// Mitsubishi GX Works2 project: NIAP1854_1000_RC-1M_5B_R3   PLC: FX3S

PROGRAM MAIN
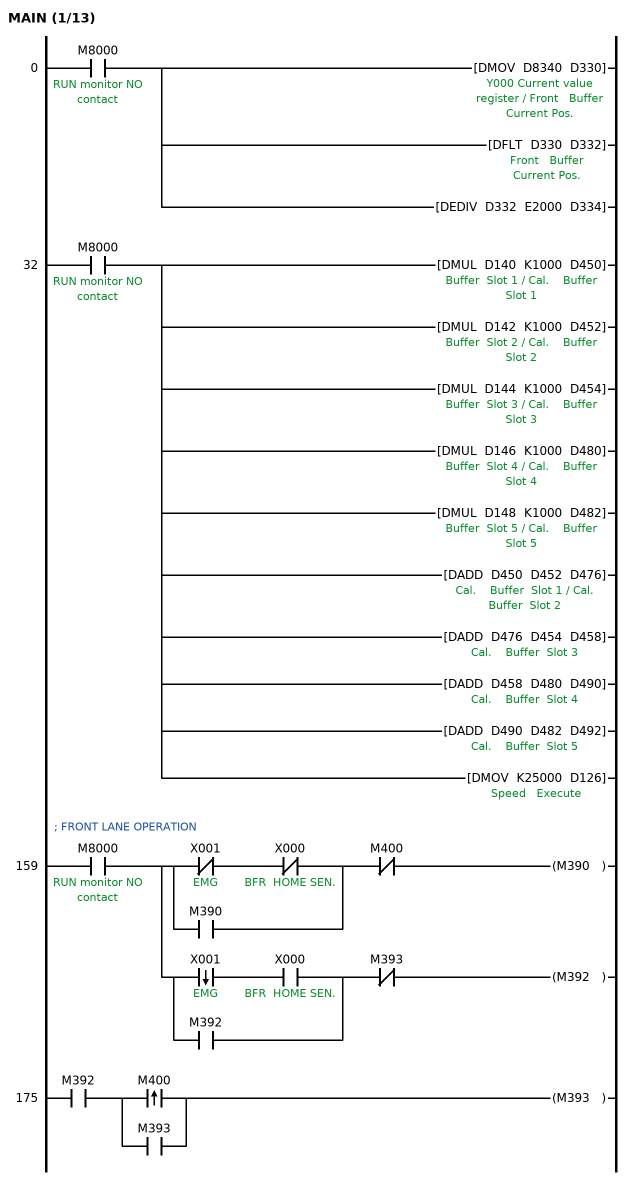
0     LD      M8000  ; RUN monitor NO contact
      DMOV    D8340 D330  ; Y000 Current value register / Front   Buffer  Current Pos.
      DFLT    D330 D332
      DEDIV   D332 E2000 D334
32    LD      M8000  ; RUN monitor NO contact
      DMUL    D140 K1000 D450  ; Buffer  Slot 1 / Cal.    Buffer  Slot 1
      DMUL    D142 K1000 D452  ; Buffer  Slot 2 / Cal.    Buffer  Slot 2
      DMUL    D144 K1000 D454  ; Buffer  Slot 3 / Cal.    Buffer  Slot 3
      DMUL    D146 K1000 D480  ; Buffer  Slot 4 / Cal.    Buffer  Slot 4
      DMUL    D148 K1000 D482  ; Buffer  Slot 5 / Cal.    Buffer  Slot 5
      DADD    D450 D452 D476
      DADD    D476 D454 D458
      DADD    D458 D480 D490
      DADD    D490 D482 D492
      DMOV    K25000 D126  ; Speed   Execute
; FRONT LANE OPERATION
159   LD      M8000  ; RUN monitor NO contact
      MPS
      LDI     X001  ; EMG
      ANI     X000  ; BFR  HOME SEN.
      OR      M390
      ANB
      ANI     M400
      OUT     M390
      MPP
      LDF     X001  ; EMG
      AND     X000  ; BFR  HOME SEN.
      OR      M392
      ANB
      ANI     M393
      OUT     M392
175   LD      M392
      LDP     M400
      OR      M393
      ANB
      OUT     M393
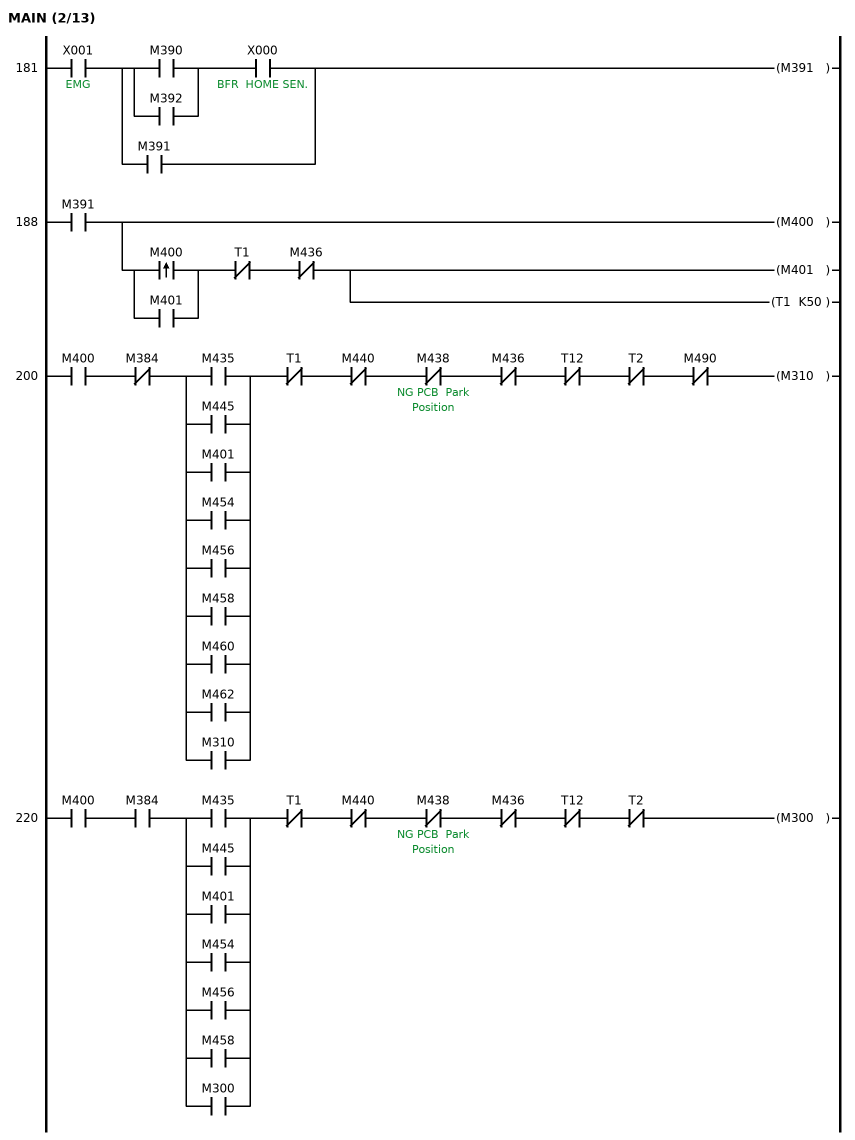
181   LD      X001  ; EMG
      LD      M390
      OR      M392
      AND     X000  ; BFR  HOME SEN.
      OR      M391
      ANB
      OUT     M391
188   LD      M391
      OUT     M400
      LDP     M400
      OR      M401
      ANB
      ANI     T1
      ANI     M436
      OUT     M401
      OUT     T1 K50
200   LD      M400
      ANI     M384
      LD      M435
      OR      M445
      OR      M401
      OR      M454
      OR      M456
      OR      M458
      OR      M460
      OR      M462
      OR      M310
      ANB
      ANI     T1
      ANI     M440
      ANI     M438  ; NG PCB  Park    Position
      ANI     M436
      ANI     T12
      ANI     T2
      ANI     M490
      OUT     M310
220   LD      M400
      AND     M384
      LD      M435
      OR      M445
      OR      M401
      OR      M454
      OR      M456
      OR      M458
      OR      M300
      ANB
      ANI     T1
      ANI     M440
      ANI     M438  ; NG PCB  Park    Position
      ANI     M436
      ANI     T12
      ANI     T2
      OUT     M300
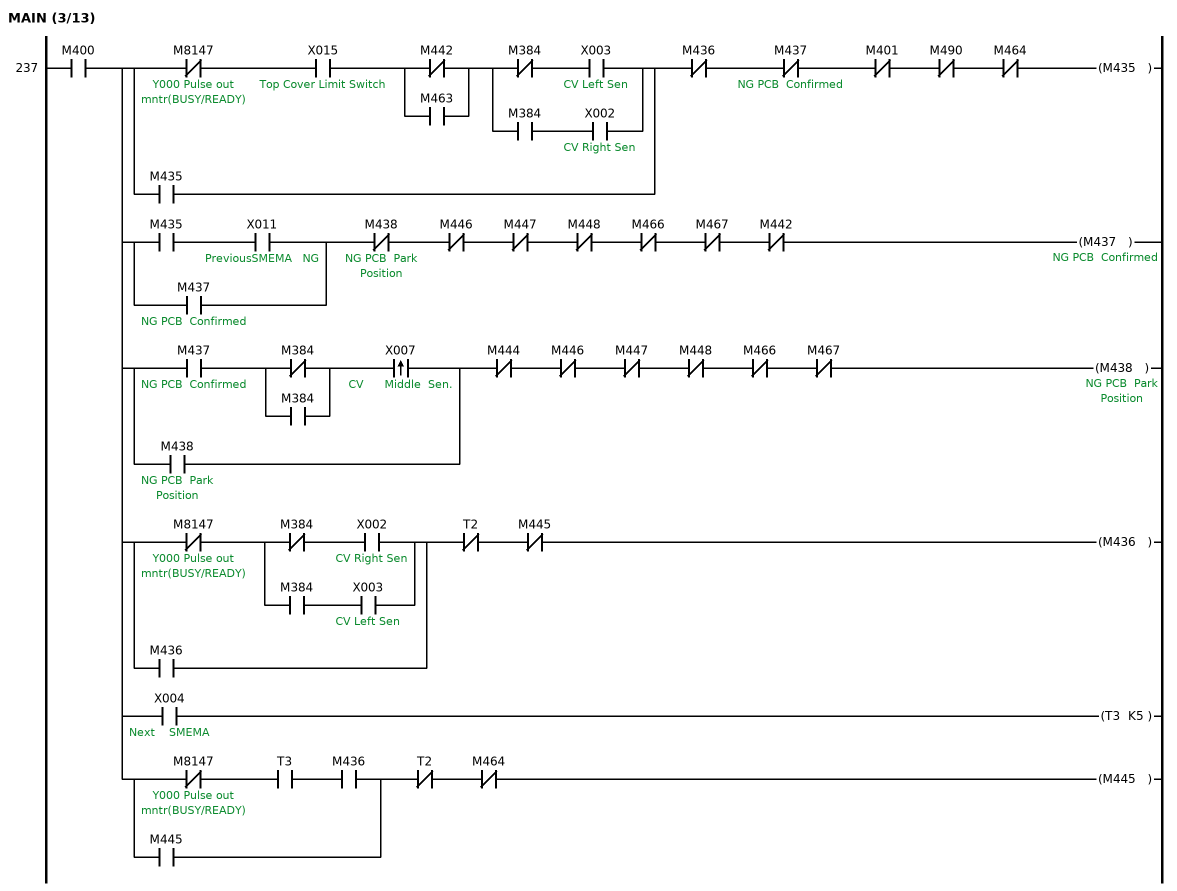
237   LD      M400
      MPS
      LDI     M8147  ; Y000 Pulse out mntr(BUSY/READY)
      AND     X015  ; Top Cover Limit Switch
      LDI     M442
      OR      M463
      ANB
      LDI     M384
      AND     X003  ; CV Left Sen
      LD      M384
      AND     X002  ; CV Right Sen
      ORB
      ANB
      OR      M435
      ANB
      ANI     M436
      ANI     M437  ; NG PCB  Confirmed
      ANI     M401
      ANI     M490
      ANI     M464
      OUT     M435
      MRD
      LD      M435
      AND     X011  ; PreviousSMEMA   NG
      OR      M437  ; NG PCB  Confirmed
      ANB
      ANI     M438  ; NG PCB  Park    Position
      ANI     M446
      ANI     M447
      ANI     M448
      ANI     M466
      ANI     M467
      ANI     M442
      OUT     M437  ; NG PCB  Confirmed
      MRD
      LD      M437  ; NG PCB  Confirmed
      LDI     M384
      OR      M384
      ANB
      ANDP    X007  ; CV      Middle  Sen.
      OR      M438  ; NG PCB  Park    Position
      ANB
      ANI     M444
      ANI     M446
      ANI     M447
      ANI     M448
      ANI     M466
      ANI     M467
      OUT     M438  ; NG PCB  Park    Position
      MRD
      LDI     M8147  ; Y000 Pulse out mntr(BUSY/READY)
      LDI     M384
      AND     X002  ; CV Right Sen
      LD      M384
      AND     X003  ; CV Left Sen
      ORB
      ANB
      OR      M436
      ANB
      ANI     T2
      ANI     M445
      OUT     M436
      MRD
      AND     X004  ; Next    SMEMA
      OUT     T3 K5
      MPP
      LDI     M8147  ; Y000 Pulse out mntr(BUSY/READY)
      AND     T3
      AND     M436
      OR      M445
      ANB
      ANI     T2
      ANI     M464
      OUT     M445
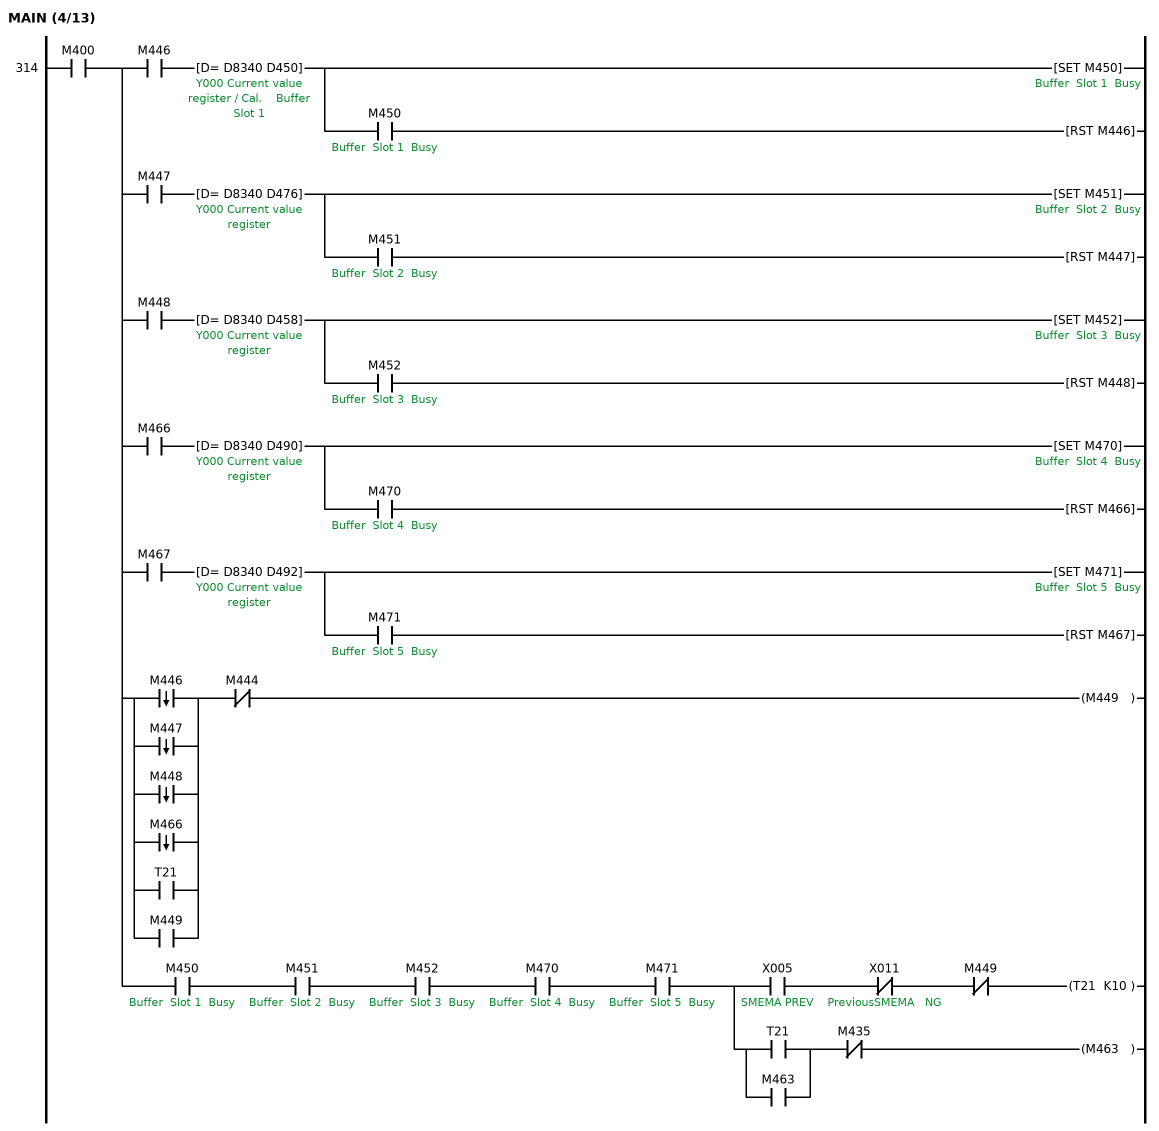
314   LD      M400
      MPS
      AND     M446
      ANDD=   D8340 D450  ; Y000 Current value register / Cal.    Buffer  Slot 1
      SET     M450  ; Buffer  Slot 1  Busy
      AND     M450  ; Buffer  Slot 1  Busy
      RST     M446
      MRD
      AND     M447
      ANDD=   D8340 D476  ; Y000 Current value register
      SET     M451  ; Buffer  Slot 2  Busy
      AND     M451  ; Buffer  Slot 2  Busy
      RST     M447
      MRD
      AND     M448
      ANDD=   D8340 D458  ; Y000 Current value register
      SET     M452  ; Buffer  Slot 3  Busy
      AND     M452  ; Buffer  Slot 3  Busy
      RST     M448
      MRD
      AND     M466
      ANDD=   D8340 D490  ; Y000 Current value register
      SET     M470  ; Buffer  Slot 4  Busy
      AND     M470  ; Buffer  Slot 4  Busy
      RST     M466
      MRD
      AND     M467
      ANDD=   D8340 D492  ; Y000 Current value register
      SET     M471  ; Buffer  Slot 5  Busy
      AND     M471  ; Buffer  Slot 5  Busy
      RST     M467
      MRD
      LDF     M446
      ORF     M447
      ORF     M448
      ORF     M466
      OR      T21
      OR      M449
      ANB
      ANI     M444
      OUT     M449
      MPP
      AND     M450  ; Buffer  Slot 1  Busy
      AND     M451  ; Buffer  Slot 2  Busy
      AND     M452  ; Buffer  Slot 3  Busy
      AND     M470  ; Buffer  Slot 4  Busy
      AND     M471  ; Buffer  Slot 5  Busy
      MPS
      AND     X005  ; SMEMA PREV
      ANI     X011  ; PreviousSMEMA   NG
      ANI     M449
      OUT     T21 K10
      MPP
      LD      T21
      OR      M463
      ANB
      ANI     M435
      OUT     M463
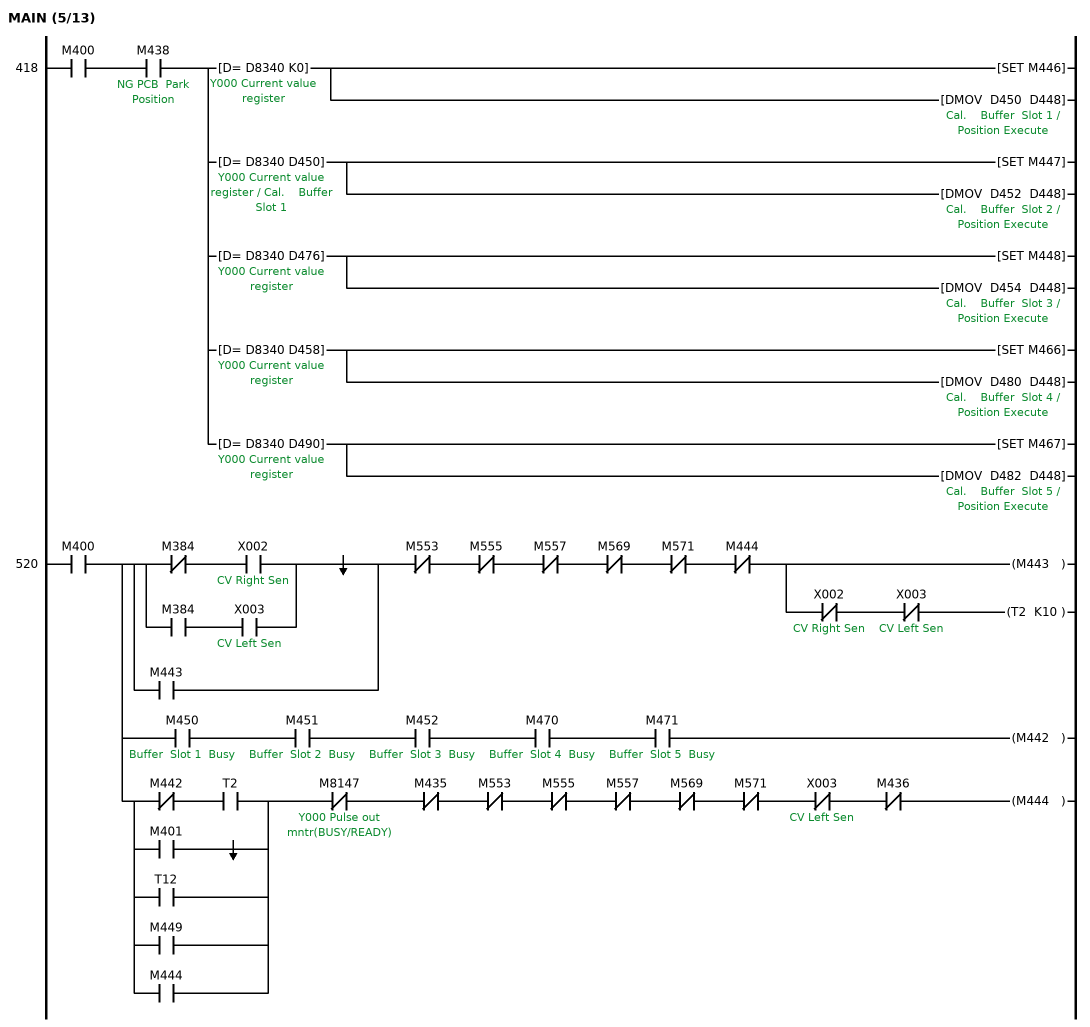
418   LD      M400
      AND     M438  ; NG PCB  Park    Position
      MPS
      ANDD=   D8340 K0  ; Y000 Current value register
      SET     M446
      DMOV    D450 D448  ; Position Execute
      MRD
      ANDD=   D8340 D450  ; Y000 Current value register / Cal.    Buffer  Slot 1
      SET     M447
      DMOV    D452 D448
      MRD
      ANDD=   D8340 D476  ; Y000 Current value register
      SET     M448
      DMOV    D454 D448
      MRD
      ANDD=   D8340 D458  ; Y000 Current value register
      SET     M466
      DMOV    D480 D448
      MPP
      ANDD=   D8340 D490  ; Y000 Current value register
      SET     M467
      DMOV    D482 D448
520   LD      M400
      MPS
      LDI     M384
      AND     X002  ; CV Right Sen
      LD      M384
      AND     X003  ; CV Left Sen
      ORB
      MEF
      OR      M443
      ANB
      ANI     M553
      ANI     M555
      ANI     M557
      ANI     M569
      ANI     M571
      ANI     M444
      OUT     M443
      ANI     X002  ; CV Right Sen
      ANI     X003  ; CV Left Sen
      OUT     T2 K10
      MRD
      AND     M450  ; Buffer  Slot 1  Busy
      AND     M451  ; Buffer  Slot 2  Busy
      AND     M452  ; Buffer  Slot 3  Busy
      AND     M470  ; Buffer  Slot 4  Busy
      AND     M471  ; Buffer  Slot 5  Busy
      OUT     M442
      MPP
      LDI     M442
      AND     T2
      LD      M401
      MEF
      ORB
      OR      T12
      OR      M449
      OR      M444
      ANB
      ANI     M8147  ; Y000 Pulse out mntr(BUSY/READY)
      ANI     M435
      ANI     M553
      ANI     M555
      ANI     M557
      ANI     M569
      ANI     M571
      ANI     X003  ; CV Left Sen
      ANI     M436
      OUT     M444
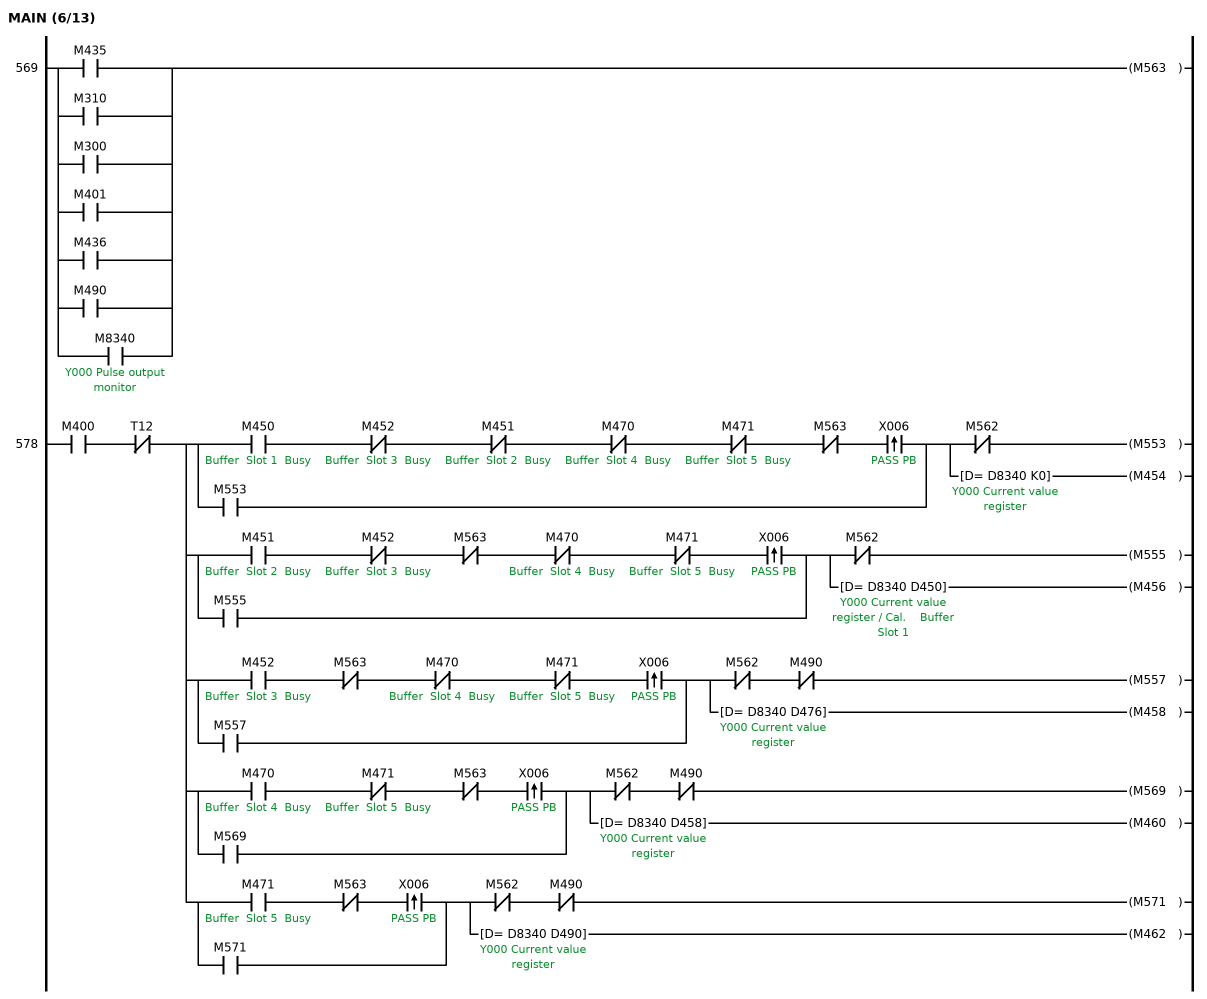
569   LD      M435
      OR      M310
      OR      M300
      OR      M401
      OR      M436
      OR      M490
      OR      M8340  ; Y000 Pulse output monitor
      OUT     M563
578   LD      M400
      ANI     T12
      MPS
      LD      M450  ; Buffer  Slot 1  Busy
      ANI     M452  ; Buffer  Slot 3  Busy
      ANI     M451  ; Buffer  Slot 2  Busy
      ANI     M470  ; Buffer  Slot 4  Busy
      ANI     M471  ; Buffer  Slot 5  Busy
      ANI     M563
      ANDP    X006  ; PASS PB
      OR      M553
      ANB
      MPS
      ANI     M562
      OUT     M553
      MPP
      ANDD=   D8340 K0  ; Y000 Current value register
      OUT     M454
      MRD
      LD      M451  ; Buffer  Slot 2  Busy
      ANI     M452  ; Buffer  Slot 3  Busy
      ANI     M563
      ANI     M470  ; Buffer  Slot 4  Busy
      ANI     M471  ; Buffer  Slot 5  Busy
      ANDP    X006  ; PASS PB
      OR      M555
      ANB
      MPS
      ANI     M562
      OUT     M555
      MPP
      ANDD=   D8340 D450  ; Y000 Current value register / Cal.    Buffer  Slot 1
      OUT     M456
      MRD
      LD      M452  ; Buffer  Slot 3  Busy
      ANI     M563
      ANI     M470  ; Buffer  Slot 4  Busy
      ANI     M471  ; Buffer  Slot 5  Busy
      ANDP    X006  ; PASS PB
      OR      M557
      ANB
      MPS
      ANI     M562
      ANI     M490
      OUT     M557
      MPP
      ANDD=   D8340 D476  ; Y000 Current value register
      OUT     M458
      MRD
      LD      M470  ; Buffer  Slot 4  Busy
      ANI     M471  ; Buffer  Slot 5  Busy
      ANI     M563
      ANDP    X006  ; PASS PB
      OR      M569
      ANB
      MPS
      ANI     M562
      ANI     M490
      OUT     M569
      MPP
      ANDD=   D8340 D458  ; Y000 Current value register
      OUT     M460
      MPP
      LD      M471  ; Buffer  Slot 5  Busy
      ANI     M563
      ANDP    X006  ; PASS PB
      OR      M571
      ANB
      MPS
      ANI     M562
      ANI     M490
      OUT     M571
      MPP
      ANDD=   D8340 D490  ; Y000 Current value register
      OUT     M462
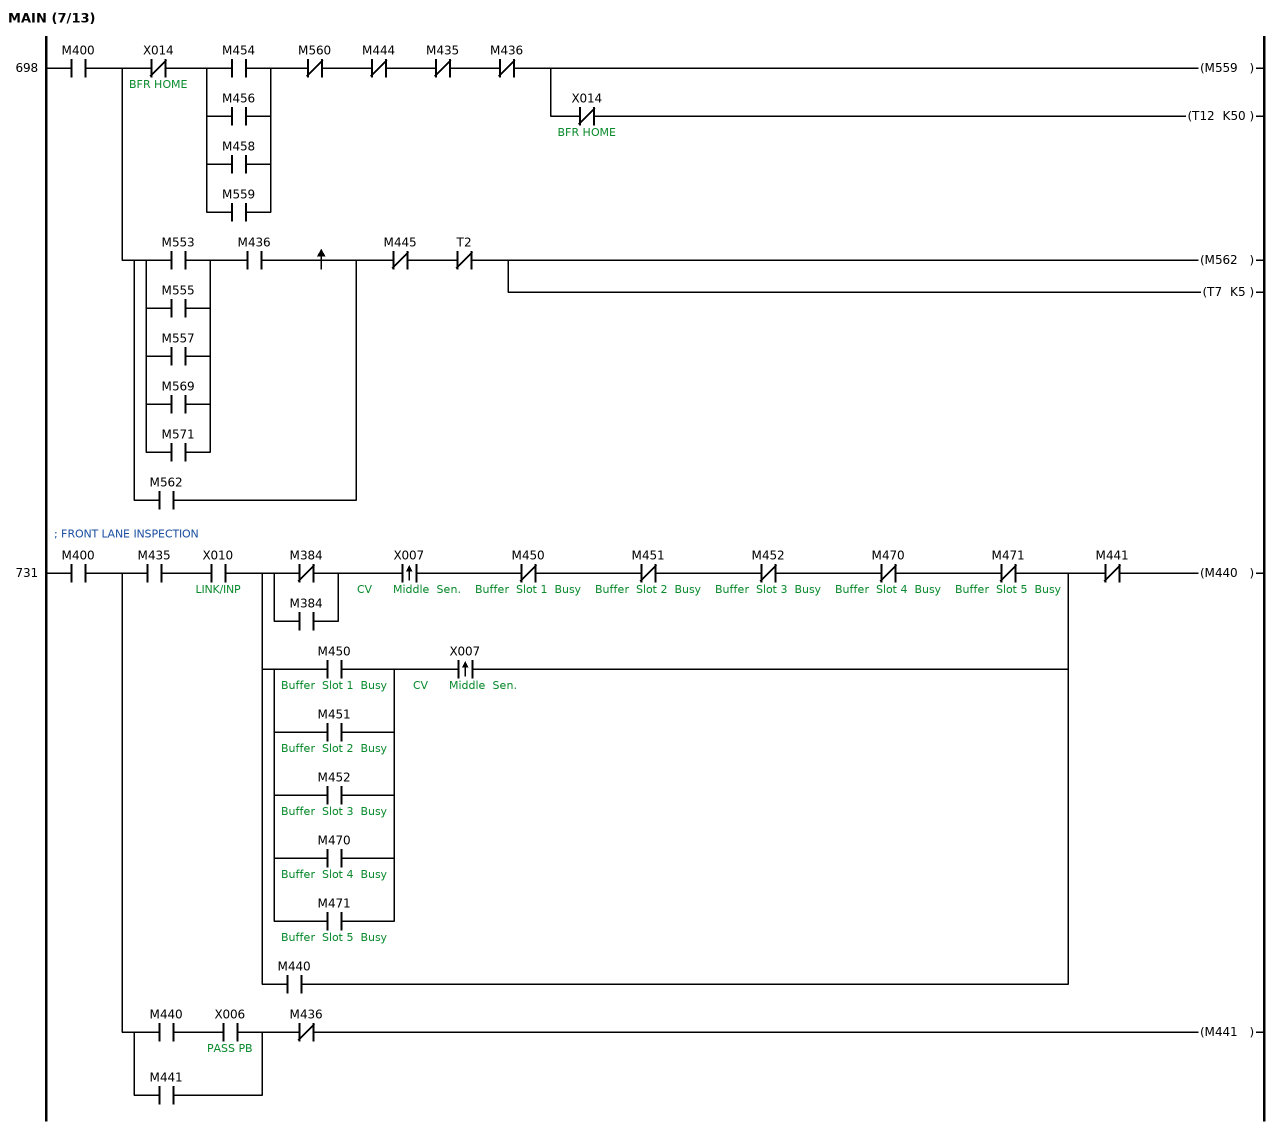
698   LD      M400
      MPS
      ANI     X014  ; BFR HOME
      LD      M454
      OR      M456
      OR      M458
      OR      M559
      ANB
      ANI     M560
      ANI     M444
      ANI     M435
      ANI     M436
      OUT     M559
      ANI     X014  ; BFR HOME
      OUT     T12 K50
      MPP
      LD      M553
      OR      M555
      OR      M557
      OR      M569
      OR      M571
      AND     M436
      MEP
      OR      M562
      ANB
      ANI     M445
      ANI     T2
      OUT     M562
      OUT     T7 K5
; FRONT LANE INSPECTION
731   LD      M400
      MPS
      AND     M435
      AND     X010  ; LINK/INP
      LDI     M384
      OR      M384
      ANDP    X007  ; CV      Middle  Sen.
      ANI     M450  ; Buffer  Slot 1  Busy
      ANI     M451  ; Buffer  Slot 2  Busy
      ANI     M452  ; Buffer  Slot 3  Busy
      ANI     M470  ; Buffer  Slot 4  Busy
      ANI     M471  ; Buffer  Slot 5  Busy
      LD      M450  ; Buffer  Slot 1  Busy
      OR      M451  ; Buffer  Slot 2  Busy
      OR      M452  ; Buffer  Slot 3  Busy
      OR      M470  ; Buffer  Slot 4  Busy
      OR      M471  ; Buffer  Slot 5  Busy
      ANDP    X007  ; CV      Middle  Sen.
      ORB
      OR      M440
      ANB
      ANI     M441
      OUT     M440
      MPP
      LD      M440
      AND     X006  ; PASS PB
      OR      M441
      ANB
      ANI     M436
      OUT     M441
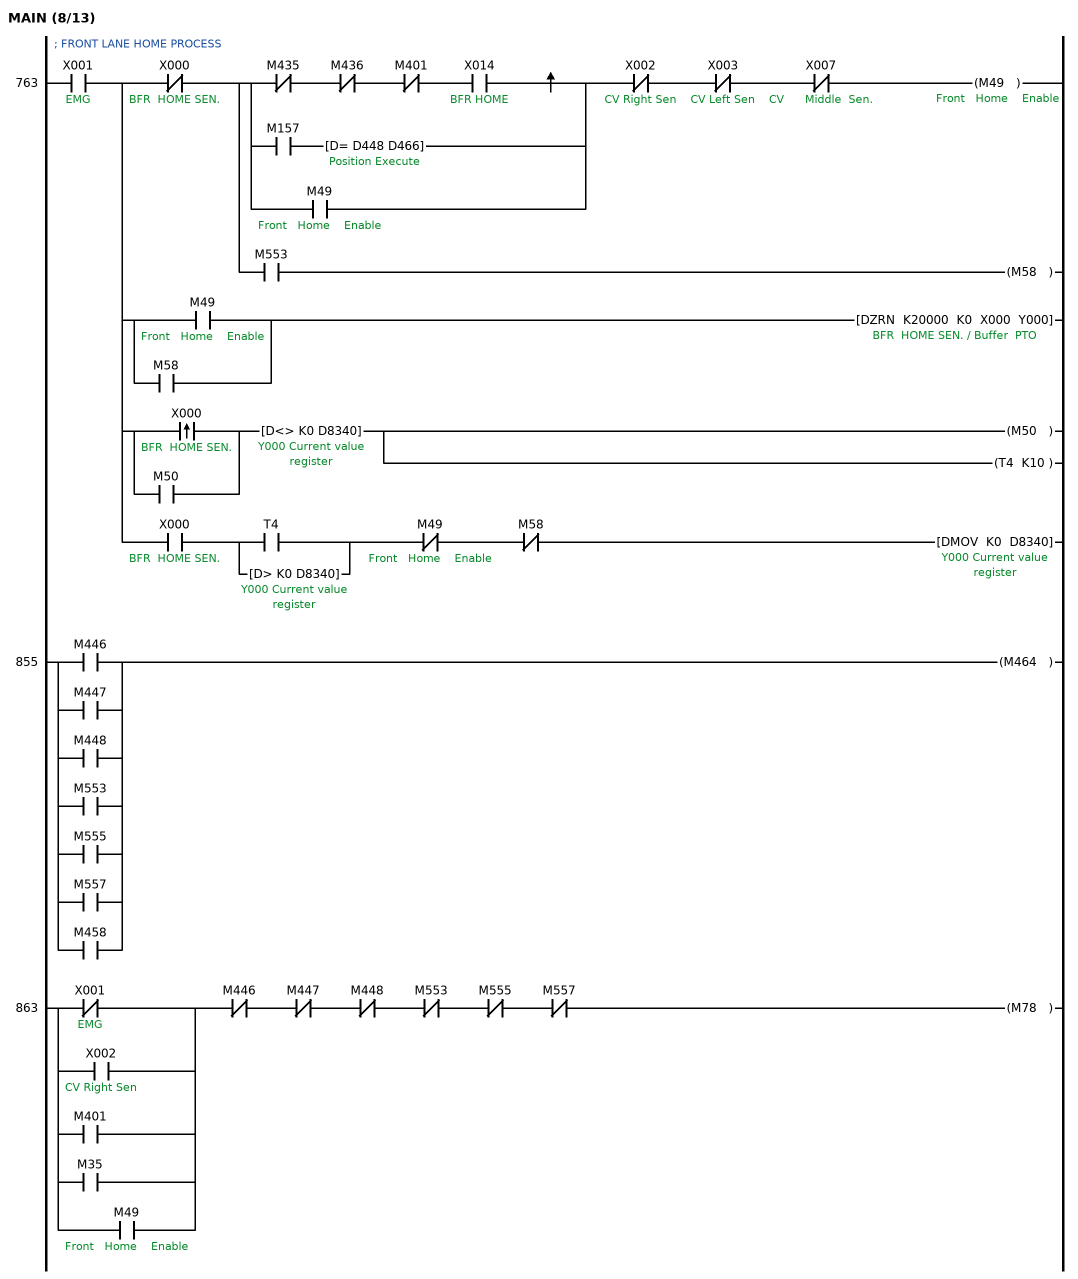
; FRONT LANE HOME PROCESS
763   LD      X001  ; EMG
      MPS
      ANI     X000  ; BFR  HOME SEN.
      MPS
      LDI     M435
      ANI     M436
      ANI     M401
      AND     X014  ; BFR HOME
      MEP
      LD      M157
      ANDD=   D448 D466  ; Position Execute
      ORB
      OR      M49  ; Front   Home    Enable
      ANB
      ANI     X002  ; CV Right Sen
      ANI     X003  ; CV Left Sen
      ANI     X007  ; CV      Middle  Sen.
      OUT     M49  ; Front   Home    Enable
      MPP
      AND     M553
      OUT     M58
      MRD
      LD      M49  ; Front   Home    Enable
      OR      M58
      ANB
      DZRN    K20000 K0 X000 Y000  ; Buffer  PTO
      MRD
      LDP     X000  ; BFR  HOME SEN.
      OR      M50
      ANB
      ANDD<>  K0 D8340  ; Y000 Current value register
      OUT     M50
      OUT     T4 K10
      MPP
      AND     X000  ; BFR  HOME SEN.
      LD      T4
      ORD>    K0 D8340  ; Y000 Current value register
      ANB
      ANI     M49  ; Front   Home    Enable
      ANI     M58
      DMOV    K0 D8340
855   LD      M446
      OR      M447
      OR      M448
      OR      M553
      OR      M555
      OR      M557
      OR      M458
      OUT     M464
863   LDI     X001  ; EMG
      OR      X002  ; CV Right Sen
      OR      M401
      OR      M35
      OR      M49  ; Front   Home    Enable
      ANI     M446
      ANI     M447
      ANI     M448
      ANI     M553
      ANI     M555
      ANI     M557
      OUT     M78
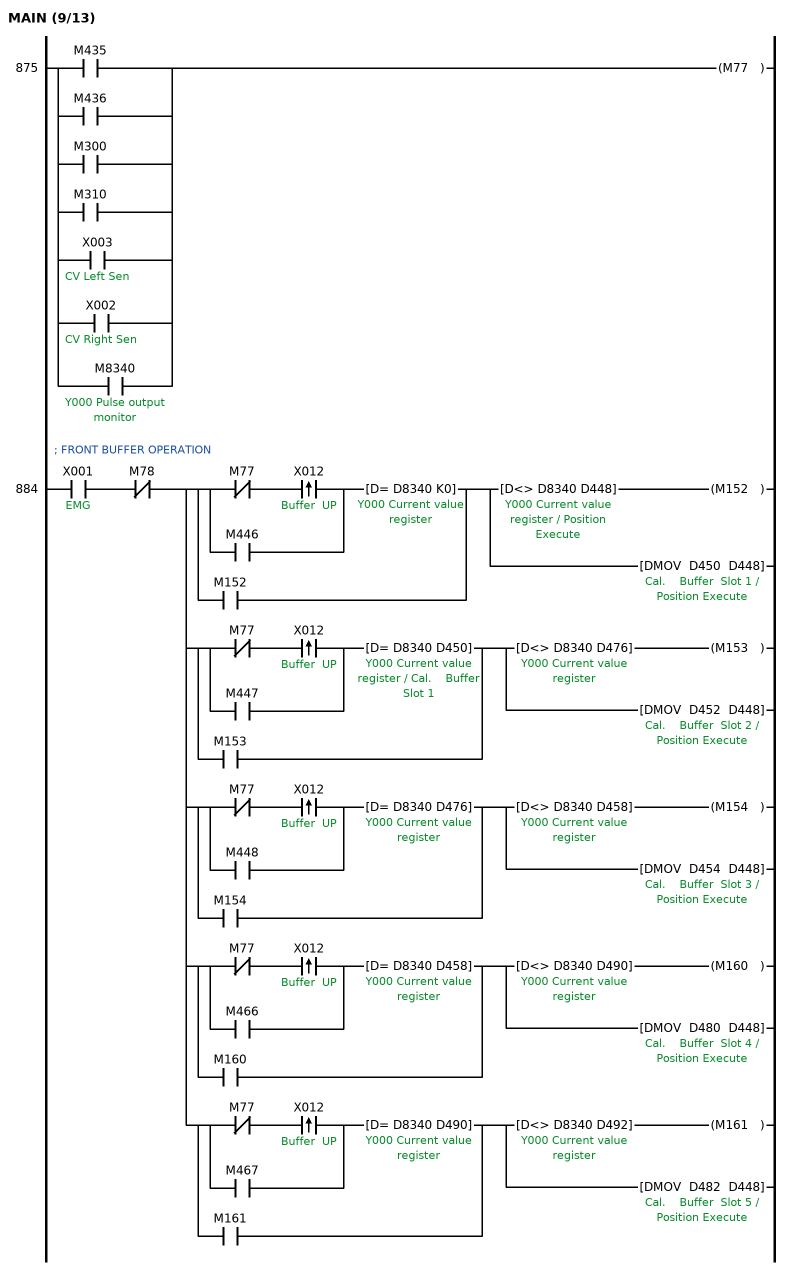
875   LD      M435
      OR      M436
      OR      M300
      OR      M310
      OR      X003  ; CV Left Sen
      OR      X002  ; CV Right Sen
      OR      M8340  ; Y000 Pulse output monitor
      OUT     M77
; FRONT BUFFER OPERATION
884   LD      X001  ; EMG
      ANI     M78
      MPS
      LDI     M77
      ANDP    X012  ; Buffer  UP
      OR      M446
      ANDD=   D8340 K0  ; Y000 Current value register
      OR      M152
      ANB
      MPS
      ANDD<>  D8340 D448  ; Y000 Current value register / Position Execute
      OUT     M152
      MPP
      DMOV    D450 D448
      MRD
      LDI     M77
      ANDP    X012  ; Buffer  UP
      OR      M447
      ANDD=   D8340 D450  ; Y000 Current value register / Cal.    Buffer  Slot 1
      OR      M153
      ANB
      MPS
      ANDD<>  D8340 D476  ; Y000 Current value register
      OUT     M153
      MPP
      DMOV    D452 D448
      MRD
      LDI     M77
      ANDP    X012  ; Buffer  UP
      OR      M448
      ANDD=   D8340 D476  ; Y000 Current value register
      OR      M154
      ANB
      MPS
      ANDD<>  D8340 D458  ; Y000 Current value register
      OUT     M154
      MPP
      DMOV    D454 D448
      MRD
      LDI     M77
      ANDP    X012  ; Buffer  UP
      OR      M466
      ANDD=   D8340 D458  ; Y000 Current value register
      OR      M160
      ANB
      MPS
      ANDD<>  D8340 D490  ; Y000 Current value register
      OUT     M160
      MPP
      DMOV    D480 D448
      MPP
      LDI     M77
      ANDP    X012  ; Buffer  UP
      OR      M467
      ANDD=   D8340 D490  ; Y000 Current value register
      OR      M161
      ANB
      MPS
      ANDD<>  D8340 D492  ; Y000 Current value register
      OUT     M161
      MPP
      DMOV    D482 D448
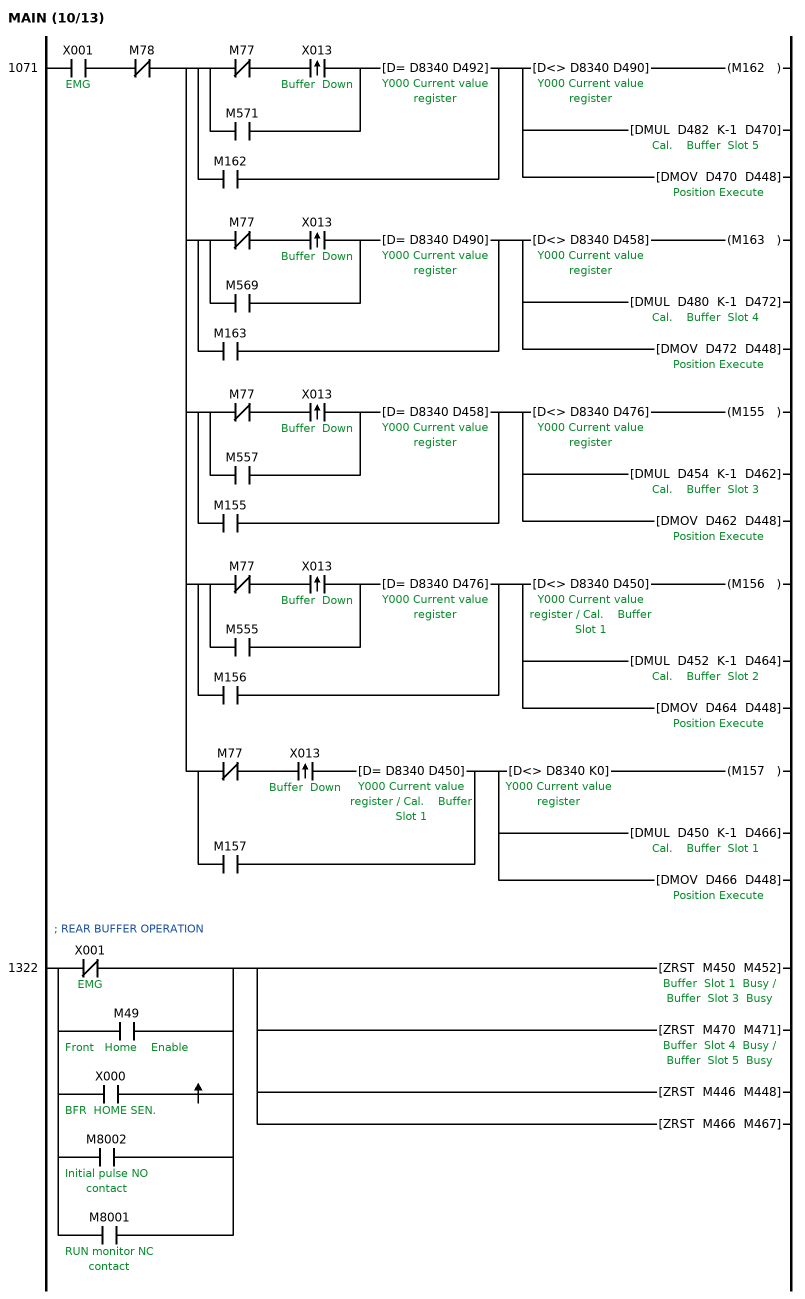
1071  LD      X001  ; EMG
      ANI     M78
      MPS
      LDI     M77
      ANDP    X013  ; Buffer  Down
      OR      M571
      ANDD=   D8340 D492  ; Y000 Current value register
      OR      M162
      ANB
      MPS
      ANDD<>  D8340 D490  ; Y000 Current value register
      OUT     M162
      MPP
      DMUL    D482 K-1 D470
      DMOV    D470 D448
      MRD
      LDI     M77
      ANDP    X013  ; Buffer  Down
      OR      M569
      ANDD=   D8340 D490  ; Y000 Current value register
      OR      M163
      ANB
      MPS
      ANDD<>  D8340 D458  ; Y000 Current value register
      OUT     M163
      MPP
      DMUL    D480 K-1 D472
      DMOV    D472 D448
      MRD
      LDI     M77
      ANDP    X013  ; Buffer  Down
      OR      M557
      ANDD=   D8340 D458  ; Y000 Current value register
      OR      M155
      ANB
      MPS
      ANDD<>  D8340 D476  ; Y000 Current value register
      OUT     M155
      MPP
      DMUL    D454 K-1 D462
      DMOV    D462 D448
      MRD
      LDI     M77
      ANDP    X013  ; Buffer  Down
      OR      M555
      ANDD=   D8340 D476  ; Y000 Current value register
      OR      M156
      ANB
      MPS
      ANDD<>  D8340 D450  ; Y000 Current value register / Cal.    Buffer  Slot 1
      OUT     M156
      MPP
      DMUL    D452 K-1 D464
      DMOV    D464 D448
      MPP
      LDI     M77
      ANDP    X013  ; Buffer  Down
      ANDD=   D8340 D450  ; Y000 Current value register / Cal.    Buffer  Slot 1
      OR      M157
      ANB
      MPS
      ANDD<>  D8340 K0  ; Y000 Current value register
      OUT     M157
      MPP
      DMUL    D450 K-1 D466
      DMOV    D466 D448
; REAR BUFFER OPERATION
1322  LDI     X001  ; EMG
      OR      M49  ; Front   Home    Enable
      LD      X000  ; BFR  HOME SEN.
      MEP
      ORB
      OR      M8002  ; Initial pulse NO contact
      OR      M8001  ; RUN monitor NC contact
      ZRST    M450 M452
      ZRST    M470 M471
      ZRST    M446 M448
      ZRST    M466 M467
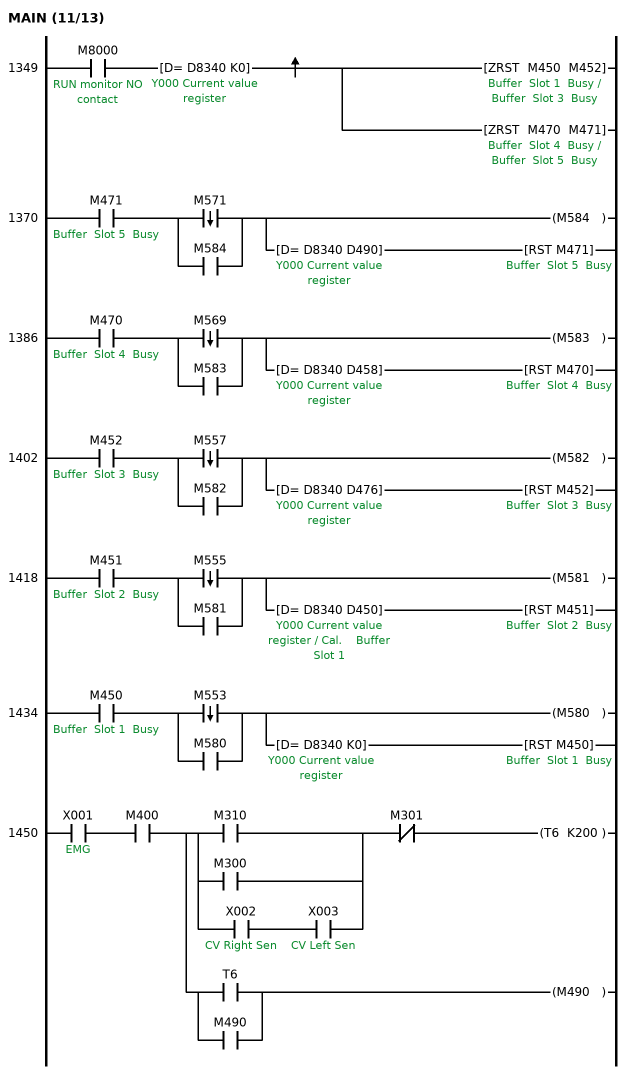
1349  LD      M8000  ; RUN monitor NO contact
      ANDD=   D8340 K0  ; Y000 Current value register
      MEP
      ZRST    M450 M452
      ZRST    M470 M471
1370  LD      M471  ; Buffer  Slot 5  Busy
      LDF     M571
      OR      M584
      ANB
      OUT     M584
      ANDD=   D8340 D490  ; Y000 Current value register
      RST     M471  ; Buffer  Slot 5  Busy
1386  LD      M470  ; Buffer  Slot 4  Busy
      LDF     M569
      OR      M583
      ANB
      OUT     M583
      ANDD=   D8340 D458  ; Y000 Current value register
      RST     M470  ; Buffer  Slot 4  Busy
1402  LD      M452  ; Buffer  Slot 3  Busy
      LDF     M557
      OR      M582
      ANB
      OUT     M582
      ANDD=   D8340 D476  ; Y000 Current value register
      RST     M452  ; Buffer  Slot 3  Busy
1418  LD      M451  ; Buffer  Slot 2  Busy
      LDF     M555
      OR      M581
      ANB
      OUT     M581
      ANDD=   D8340 D450  ; Y000 Current value register / Cal.    Buffer  Slot 1
      RST     M451  ; Buffer  Slot 2  Busy
1434  LD      M450  ; Buffer  Slot 1  Busy
      LDF     M553
      OR      M580
      ANB
      OUT     M580
      ANDD=   D8340 K0  ; Y000 Current value register
      RST     M450  ; Buffer  Slot 1  Busy
1450  LD      X001  ; EMG
      AND     M400
      MPS
      LD      M310
      OR      M300
      LD      X002  ; CV Right Sen
      AND     X003  ; CV Left Sen
      ORB
      ANB
      ANI     M301
      OUT     T6 K200
      MPP
      LD      T6
      OR      M490
      ANB
      OUT     M490
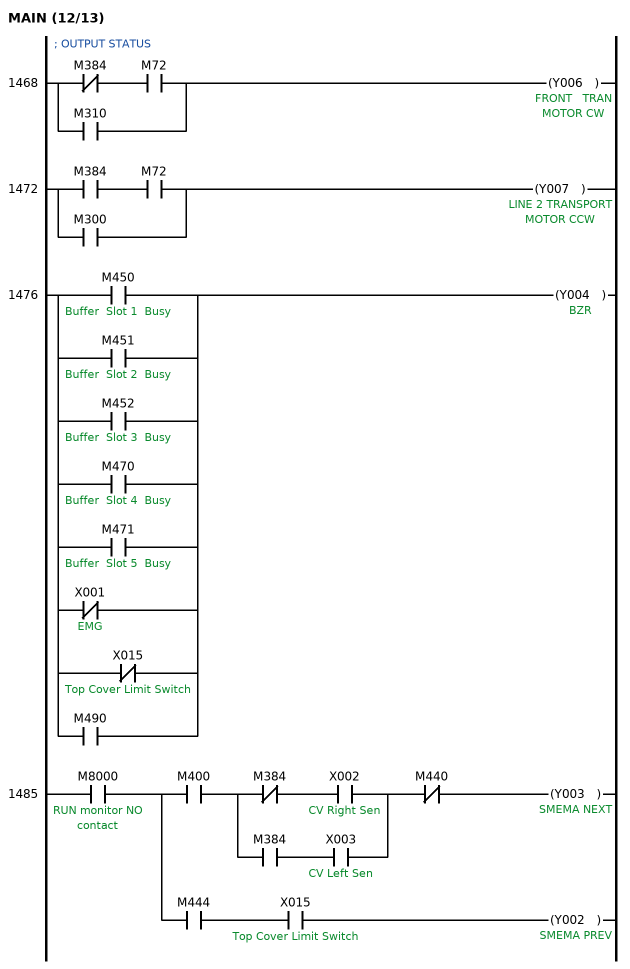
; OUTPUT STATUS
1468  LDI     M384
      AND     M72
      OR      M310
      OUT     Y006  ; FRONT   TRAN    MOTOR CW
1472  LD      M384
      AND     M72
      OR      M300
      OUT     Y007  ; LINE 2 TRANSPORT MOTOR CCW
1476  LD      M450  ; Buffer  Slot 1  Busy
      OR      M451  ; Buffer  Slot 2  Busy
      OR      M452  ; Buffer  Slot 3  Busy
      OR      M470  ; Buffer  Slot 4  Busy
      OR      M471  ; Buffer  Slot 5  Busy
      ORI     X001  ; EMG
      ORI     X015  ; Top Cover Limit Switch
      OR      M490
      OUT     Y004  ; BZR
1485  LD      M8000  ; RUN monitor NO contact
      MPS
      AND     M400
      LDI     M384
      AND     X002  ; CV Right Sen
      LD      M384
      AND     X003  ; CV Left Sen
      ORB
      ANB
      ANI     M440
      OUT     Y003  ; SMEMA NEXT
      MPP
      AND     M444
      AND     X015  ; Top Cover Limit Switch
      OUT     Y002  ; SMEMA PREV
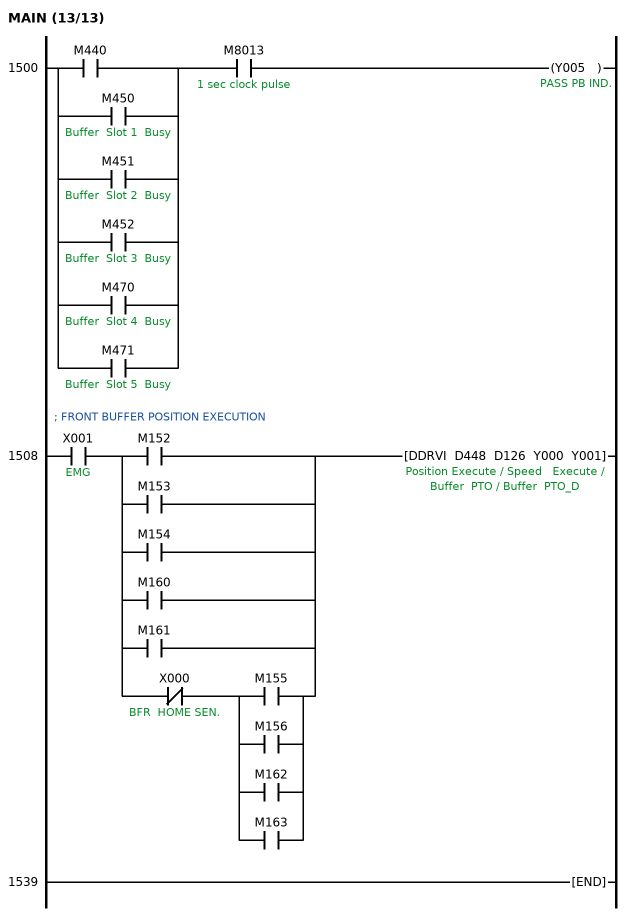
1500  LD      M440
      OR      M450  ; Buffer  Slot 1  Busy
      OR      M451  ; Buffer  Slot 2  Busy
      OR      M452  ; Buffer  Slot 3  Busy
      OR      M470  ; Buffer  Slot 4  Busy
      OR      M471  ; Buffer  Slot 5  Busy
      AND     M8013  ; 1 sec clock pulse
      OUT     Y005  ; PASS PB IND.
; FRONT BUFFER POSITION EXECUTION
1508  LD      X001  ; EMG
      LD      M152
      OR      M153
      OR      M154
      OR      M160
      OR      M161
      LDI     X000  ; BFR  HOME SEN.
      LD      M155
      OR      M156
      OR      M162
      OR      M163
      ANB
      ORB
      ANB
      DDRVI   D448 D126 Y000 Y001  ; Buffer  PTO_D
1539  END
END_PROGRAM

// device comments not shown above
M700  ; FRONT   OPERATION
M750  ; F. BFR  SLOT 1  BUSY
M751  ; F. BFR  SLOT 2  BUSY
M752  ; F. BFR  SLOT 3  BUSY
M790  ; FRONT   PCB TRF ERROR
M791  ; REAR    PCB TRF ERROR
M850  ; R. BFR  SLOT 1  BUSY
M851  ; F. BFR  SLOT 2  BUSY
M852  ; F. BFR  SLOT 3  BUSY
D600  ; FRONT   BFR_1
D602  ; FRONT   BFR_2
D604  ; FRONT   BFR_3
D606  ; REAR    BFR_1
D608  ; REAR    BFR_2
D610  ; REAR    BFR_3
D826  ; BFR     SPEED
D848  ; FRONT   BFR EXE.POS
D1030  ; FRONT   BFR     CURRENT
